Staubli VAL3: cycle_waitEmpty.pgx

program cycle_waitEmpty()
begin
  // MOTION
  waitEndMove()
  wait(isEmpty())
  // task event
  call action_wait()
  // set the last time measure
  cycleStatus:nLastTimer=clock()-cycleStatus:nClockAction
end
